FUNCTION_BLOCK PUBLIC ElmoBasicAxis_FB EXTENDS CoE_BasicAxis_FB  
VAR_INPUT		
	pDigIn: 		    POINTER TO DINT;
	
END_VAR
VAR_IN_OUT	
END_VAR
VAR_OUTPUT	
END_VAR

VAR
	
	fbElmoIOsHandle:	FB_ElmoIOsHandle;
END_VAR


AxisCtrlPtr^.Input.Parameter.Drive.eDriveType := enumDriveType.eElmo;	
AxisCtrlPtr^.Input.Parameter.Drive.VendorNameID := eVendorNameID.Elmo;
SUPER^(AxisRef:=AxisRef);


IF pDigIn <> 0 THEN
	fbElmoIOsHandle(DigIn:=	pDigIn^);
	AxisCtrlPtr^.Output.Status.DriveEnable:=	fbElmoIOsHandle.bEnable;
END_IF

METHOD CreateDriveErrMsgDetails : enumMotorEvents
VAR_INPUT
	ErrorId			: UDINT;
END_VAR
CASE ErrorId OF
	16#0:
		CreateDriveErrMsgDetails := enumMotorEvents.NoEvents;
		
	16#2340:
		CreateDriveErrMsgDetails := enumMotorEvents.MotorSupplyError;
		fnLogMsg(ADR(LogMsg_0),LOG_ERROR,'Elmo Drive ErrorId %d  ,Short circuit',UDINT_TO_DINT(ErrorId),0,0);
	16#3120: 
		CreateDriveErrMsgDetails := enumMotorEvents.MotorSupplyError;
		fnLogMsg(ADR(LogMsg_0),LOG_ERROR,'Elmo Drive ErrorId %d Under Voltage',UDINT_TO_DINT(ErrorId),0,0);
	16#3130:
		CreateDriveErrMsgDetails := enumMotorEvents.MotorSupplyError;
		fnLogMsg(ADR(LogMsg_0),LOG_ERROR,'Elmo Drive ErrorId %d Hall  AC fail,loss off phase',UDINT_TO_DINT(ErrorId),0,0);
	16#3310:
		CreateDriveErrMsgDetails := enumMotorEvents.MotorOverCurrent ;
		fnLogMsg(ADR(LogMsg_0),LOG_ERROR,' voltage is too high',UDINT_TO_DINT(ErrorId),0,0);
 
	16#4310:
		CreateDriveErrMsgDetails := enumMotorEvents.MotorOverTemp ;
		fnLogMsg(ADR(LogMsg_0),LOG_ERROR,'Elmo Drive ErrorId %d Temp drive overhating',UDINT_TO_DINT(ErrorId),0,0);
	16#5280:
		CreateDriveErrMsgDetails := enumMotorEvents.MotorPositionError ;	
		fnLogMsg(ADR(LogMsg_0),LOG_ERROR,'Elmo Drive ErrorId %d Gantry position error',UDINT_TO_DINT(ErrorId),0,0);
		
	16#5441:
		CreateDriveErrMsgDetails := enumMotorEvents.DriveNotEnabled;
		fnLogMsg(ADR(LogMsg_0),LOG_ERROR,'Elmo Drive ErrorId %d Motor disables',UDINT_TO_DINT(ErrorId),0,0);
	16#5442:
		CreateDriveErrMsgDetails := enumMotorEvents.DriveNotEnabled;
		fnLogMsg(ADR(LogMsg_0),LOG_ERROR,'Elmo Drive ErrorId %d Motor disables by sw',UDINT_TO_DINT(ErrorId),0,0);
	16#6300:
		CreateDriveErrMsgDetails := enumMotorEvents.PLCIllegalParam;
		fnLogMsg(ADR(LogMsg_0),LOG_ERROR,'Elmo Drive ErrorId %d RPDO failed',UDINT_TO_DINT(ErrorId),0,0);
	16#7121:
		CreateDriveErrMsgDetails := enumMotorEvents.MotorPositionError;
		fnLogMsg(ADR(LogMsg_0),LOG_ERROR,'Elmo Drive ErrorId %d Motor stuck',UDINT_TO_DINT(ErrorId),0,0);
	16#7300:
		CreateDriveErrMsgDetails := enumMotorEvents.MotorFeedBackErr;
		fnLogMsg(ADR(LogMsg_0),LOG_ERROR,'Elmo Drive ErrorId %d Feedback error',UDINT_TO_DINT(ErrorId),0,0);
	16#7381:
 		CreateDriveErrMsgDetails := enumMotorEvents.DriveComError;
		fnLogMsg(ADR(LogMsg_0),LOG_ERROR,'Elmo Drive ErrorId %d 2 Dig halls sens where cng on the same time',UDINT_TO_DINT(ErrorId),0,0);
	16#7382: 
		CreateDriveErrMsgDetails := enumMotorEvents.MotorPositionError;
		fnLogMsg(ADR(LogMsg_0),LOG_ERROR,'Elmo Drive ErrorId %d Commutaition procees failed',UDINT_TO_DINT(ErrorId),0,0);
	16#8110:
		CreateDriveErrMsgDetails := enumMotorEvents.DriveComError;
		fnLogMsg(ADR(LogMsg_0),LOG_ERROR,'Elmo Drive ErrorId %d Cam Msg lost',UDINT_TO_DINT(ErrorId),0,0);
	16#8130:
		CreateDriveErrMsgDetails := enumMotorEvents.DriveComError;
		fnLogMsg(ADR(LogMsg_0),LOG_ERROR,'Elmo Drive ErrorId %d Heartbeat event',UDINT_TO_DINT(ErrorId),0,0);
	16#8140:
		CreateDriveErrMsgDetails := enumMotorEvents.MotorGeneralError;
		fnLogMsg(ADR(LogMsg_0),LOG_ERROR,'Elmo Drive ErrorId %d Recovered from bus off',UDINT_TO_DINT(ErrorId),0,0);
	16#8210:
		CreateDriveErrMsgDetails := enumMotorEvents.MotorGeneralError;
		fnLogMsg(ADR(LogMsg_0),LOG_ERROR,'Elmo Drive ErrorId %d access to non configured PDO',UDINT_TO_DINT(ErrorId),0,0);
	16#8311:
		CreateDriveErrMsgDetails := enumMotorEvents.MotorOverCurrent;
		fnLogMsg(ADR(LogMsg_0),LOG_ERROR,'Elmo Drive ErrorId %d Peak current has been exceeded',UDINT_TO_DINT(ErrorId),0,0);

	16#8480:
		CreateDriveErrMsgDetails := enumMotorEvents.MotorSpeedError;
		fnLogMsg(ADR(LogMsg_0),LOG_ERROR,'Elmo Drive ErrorId %d speed tracking Error',UDINT_TO_DINT(ErrorId),0,0);
	16#8481:
		CreateDriveErrMsgDetails := enumMotorEvents.MotorSpeedError;
		fnLogMsg(ADR(LogMsg_0),LOG_ERROR,'Elmo Drive ErrorId %d Speed limit Exceeded',UDINT_TO_DINT(ErrorId),0,0);
	16#8611:
		CreateDriveErrMsgDetails := enumMotorEvents.MotorPositionError;
		fnLogMsg(ADR(LogMsg_0),LOG_ERROR,'Elmo Drive ErrorId %d Position tracking error',UDINT_TO_DINT(ErrorId),0,0);
	16#8680:
		CreateDriveErrMsgDetails := enumMotorEvents.MotorPositionError;
		fnLogMsg(ADR(LogMsg_0),LOG_ERROR,'Elmo Drive ErrorId %d Position limit Exceeded',UDINT_TO_DINT(ErrorId),0,0);
	16#FF02:
		CreateDriveErrMsgDetails := enumMotorEvents.DriveComError;
		fnLogMsg(ADR(LogMsg_0),LOG_ERROR,'Elmo Drive ErrorId %d Com Error',UDINT_TO_DINT(ErrorId),0,0);
	16#FF10:
		CreateDriveErrMsgDetails := enumMotorEvents.MotorGeneralError ;
		fnLogMsg(ADR(LogMsg_0),LOG_ERROR,'Elmo Drive ErrorId %d Failed to start motor',UDINT_TO_DINT(ErrorId),0,0);
	16#FF20:
		CreateDriveErrMsgDetails := enumMotorEvents.MotorGeneralError;
		fnLogMsg(ADR(LogMsg_0),LOG_ERROR,'Elmo Drive ErrorId %d Saftey torque Off in use',UDINT_TO_DINT(ErrorId),0,0);
	16#FF40:
		CreateDriveErrMsgDetails := enumMotorEvents.MotorGeneralError;
		fnLogMsg(ADR(LogMsg_0),LOG_ERROR,'Elmo Drive ErrorId %d Gantry slave Disabled',UDINT_TO_DINT(ErrorId),0,0);
	ELSE
		fnLogMsg(ADR(LogMsg_0),LOG_ERROR,'unknown Elmo Drive ErrorId %d ',UDINT_TO_DINT(ErrorId),0,0);
		CreateDriveErrMsgDetails := enumMotorEvents.MotorGeneralError;
		 
END_CASE
END_METHOD

METHOD DriveUnitsTorqueToRealValue : LREAL
VAR_INPUT
	
	Torque: LREAL;	

END_VAR
DriveUnitsTorqueToRealValue := (Torque*AxisCtrlPtr^.Input.Parameter.RatedCurrent)/1000;
END_METHOD

METHOD GetCanOpenAdr : BOOL
VAR_INPUT
END_VAR


VAR
	
	SpeedSwSubIndex: INT;
END_VAR
    SUPER^.GetCanOpenAdr();	

	
	CoEDrive_Ctrl_Adr.KpSpeed.Index	   := 16#3113;	
	CoEDrive_Ctrl_Adr.KpSpeed.SunIndex  := 2;
	CoEDrive_Ctrl_Adr.KpSpeed.Size      := 4;
	CoEDrive_Ctrl_Adr.KpSpeed.IsReal    := TRUE;
	
	
	CoEDrive_Ctrl_Adr.KiSpeed.Index	    := 16#310C;	
	CoEDrive_Ctrl_Adr.KiSpeed.SunIndex  := 2;
   	CoEDrive_Ctrl_Adr.KiSpeed.Size      := 4;
	CoEDrive_Ctrl_Adr.KiSpeed.IsReal    := TRUE;
	
	CoEDrive_Ctrl_Adr.GainScheduler.Index	    := 16#30AE;	
	CoEDrive_Ctrl_Adr.GainScheduler.SunIndex    := 2;
   	CoEDrive_Ctrl_Adr.GainScheduler.Size        := 8;
	
	
	CoEDrive_Ctrl_Adr.AccClosePosErr.Index	    := 16#30AE;	
	CoEDrive_Ctrl_Adr.AccClosePosErr.SunIndex    := 9;
   	CoEDrive_Ctrl_Adr.AccClosePosErr.Size        := 8;
END_METHOD

METHOD GetErrCanAdr : BOOL
VAR_INPUT
END_VAR


VAR
	
END_VAR

	
	CoeErrIdIndex	 := 16#603F;
	CoeErrIdSubIndex := 0;
END_METHOD

METHOD  INIT_Specific : BOOL 
VAR_INPUT
	bStart: 					BOOL;
END_VAR
VAR_INST	
	ComDelay:	TON;
	Elmo_Init_State : INT ;
	ExecuteTrig: 	Trigger;
END_VAR
IF ExecuteTrig.EDGEPOS(bStart) THEN
	INIT_Specific := FALSE ;
	IF AxisCtrlPtr^.Input.Parameter.Drive.bDisableFoE_Transfer THEN 
		Elmo_Init_State:= 3;
	ELSE
		CoEDrive_Ctrl_Adr.ParamsVersionObj.Index    := 16#2F00;
		CoEDrive_Ctrl_Adr.ParamsVersionObj.SunIndex := 1; 		
		Elmo_Init_State:= 1;
	END_IF
END_IF


IF ExecuteTrig.EDGENEG(bStart) THEN
	Elmo_Init_State := 0;
END_IF	

	
CASE Elmo_Init_State OF							
	1:
		Meth_UpdateDriveParams(FALSE);
		Elmo_Init_State:=	2;
	2:	
		IF Meth_UpdateDriveParams(TRUE) THEN
			Elmo_Init_State:=	3;
		ELSIF AxisCtrlPtr^.Output.Status.Drive.eUpdate_Staus = enum_DriveUpdateStatus.Error THEN
			//
		END_IF

	3:
		ReadInitDriveParID(FALSE);
		Elmo_Init_State:=	4;
		
	4:
		IF ReadInitDriveParID(TRUE) THEN
			Elmo_Init_State:=	10;
		END_IF			

	10:
		
		Elmo_Init_State := 0 ;
		INIT_Specific := TRUE ;
		AxisCtrlPtr^.Output.Status.AxisInitDone := TRUE ;
		AxisCtrlPtr^.Output.Status.ReadyForCmd := TRUE ;
END_CASE
END_METHOD

METHOD Meth_ChangingOperationMode : BOOL
VAR_INPUT
	Execute   : BOOL;
	OperMode : eDriveModeOfOperation; 
	
END_VAR
VAR_INST
	
	ElmoCngOperState : INT;	
END_VAR

VAR
	
	ChangeDone : BOOL;
END_VAR
IF ChangeModeOperTrig.EDGEPOS(Execute) THEN

	Meth_ChangingOperationMode := FALSE;					
	ChangeDone := FALSE;
	ElmoCngOperState := 1;

	
END_IF


IF ChangeModeOperTrig.EDGENEG(Execute) THEN
	
	ElmoCngOperState := 0;
END_IF



CASE ElmoCngOperState OF
	0:
		Meth_CoEChangOperationMode(FALSE,eCaOpDriveModeOfOperation.ProfilePositionMode);
		
	1: 
		//Meth_CoEChangOperationMode
		CASE OperMode OF
			eDriveModeOfOperation.ProfilePositionMode				:
				IF Meth_CoEChangOperationMode(TRUE,eCaOpDriveModeOfOperation.ProfilePositionMode) THEN
					ChangeDone := TRUE;
				END_IF
				
		    eDriveModeOfOperation.VelocityCtrMode    				:
				IF Meth_CoEChangOperationMode(TRUE,eCaOpDriveModeOfOperation.ProfileVelocityMode)THEN
					ChangeDone := TRUE;
				END_IF
		    eDriveModeOfOperation.ProfileVelocityMode 	   	    :
				IF Meth_CoEChangOperationMode(TRUE,eCaOpDriveModeOfOperation.ProfileVelocityMode) THEN
					ChangeDone := TRUE;
				END_IF
				
		    eDriveModeOfOperation.TorqueVelocityMode 				:
				IF Meth_CoEChangOperationMode(TRUE,eCaOpDriveModeOfOperation.TorqueVelocityMode) THEN
					ChangeDone := TRUE;
				END_IF
				
		    eDriveModeOfOperation.HomingMode				    	:
				IF Meth_CoEChangOperationMode(TRUE,eCaOpDriveModeOfOperation.HomingMode)THEN
					ChangeDone := TRUE;
				END_IF
				
		    eDriveModeOfOperation.InterpolationPosMode			:
				IF Meth_CoEChangOperationMode(TRUE,eCaOpDriveModeOfOperation.InterpolationPosMode) THEN
					ChangeDone := TRUE;
				END_IF
		    eDriveModeOfOperation.CyclicSyncMode					:
				Meth_CoEChangOperationMode(TRUE,eCaOpDriveModeOfOperation.CyclicSyncMode);
		END_CASE
		ElmoCngOperState := 2;

	2:
 		Meth_ChangingOperationMode := TRUE;
		
		
END_CASE
END_METHOD

METHOD Meth_TorqueInDriveUnits : LREAL
VAR_INPUT
	
	Torque: LREAL;	

END_VAR
IF AxisCtrlPtr^.Input.Parameter.RatedCurrent <> 0 THEN
	Meth_TorqueInDriveUnits := (Torque*1000)/AxisCtrlPtr^.Input.Parameter.RatedCurrent;
END_IF
END_METHOD

METHOD ReadActualCurrent : LREAL
VAR_INPUT
END_VAR
VAR_INST
		
END_VAR


// Units [rms]

AxisCtrlPtr^.Output.monitor.ActualCurrent	:=  ( (THIS^.io_ActualCurrent) / 1000.0) * AxisCtrlPtr^.Input.Parameter.RatedCurrent / SQRT(2.0);
END_METHOD

METHOD ReadActualTorque : LREAL
VAR_INPUT
END_VAR
VAR_INST
		
END_VAR

// Units [rms]
//AxisCtrlPtr^.Output.monitor.ActualCurrent Get from ReadActualCurrent method
// on Elmo it is needed to link only IO  io_ActualCurrent
AxisCtrlPtr^.Output.monitor.ActualTorque	:=  AxisCtrlPtr^.Output.monitor.ActualCurrent * AxisCtrlPtr^.Input.Parameter.Drive.Kt;
END_METHOD

METHOD ReadInitDriveParID : BOOL
VAR_INPUT
	bStart : BOOL;
END_VAR

VAR_INST
	ExecuteTrig_1: 		Trigger;
	State_InitSpecific_1: INT;
END_VAR

IF ExecuteTrig_1.EDGEPOS(bStart) THEN
	ReadInitDriveParID		:= FALSE;
	State_InitSpecific_1	:= 1;		
END_IF

IF ExecuteTrig_1.EDGENEG(bStart) THEN
	State_InitSpecific_1	:= 0;	
	ReadInitDriveParID		:= FALSE;
END_IF

CASE State_InitSpecific_1 OF

	 
	
	1:
		SUPER^.EcCoeSdoRead(FALSE);
		CoeSdoRW.Input.Read.nIndex		:= DINT_TO_WORD(eElmoDriveParID.RatedCurrent);
		CoeSdoRW.Input.Read.nSubIndex	:= 0;
		CoeSdoRW.Input.Read.pDstBuf		:= ADR(CoeRead_RatedCurrent);
		CoeSdoRW.Input.Read.cbBufLen	:= SIZEOF(CoeRead_RatedCurrent);
		State_InitSpecific_1	:= 2;
		
	2:
		IF SUPER^.EcCoeSdoRead(TRUE) THEN	
			State_InitSpecific_1	:= 3;
		END_IF
		
	3:
		SUPER^.EcCoeSdoRead(FALSE);
		CoeSdoRW.Input.Read.nIndex		:= DINT_TO_WORD(eElmoDriveParID.RatedTorque);
		CoeSdoRW.Input.Read.nSubIndex	:= 0;
		CoeSdoRW.Input.Read.pDstBuf		:= ADR(CoeRead_RatedTorque);
		CoeSdoRW.Input.Read.cbBufLen	:= SIZEOF(CoeRead_RatedTorque);
		State_InitSpecific_1	:= 4;
		
	4:
		IF SUPER^.EcCoeSdoRead(TRUE) THEN
			AxisCtrlPtr^.Input.Parameter.RatedCurrent	:= UDINT_TO_LREAL(CoeRead_RatedCurrent) / 1000.0;
			AxisCtrlPtr^.Input.Parameter.Ratedtorque	:= UDINT_TO_LREAL(CoeRead_RatedTorque) / 1000.0;
			ReadInitDriveParID		:= TRUE;	
			State_InitSpecific_1	:= 0;
		END_IF
		
END_CASE
END_METHOD

END_FUNCTION_BLOCK

(* stored: Version 1.1.0.1, ProductVersion 3.1.4024.3
   POU ElmoBasicAxis_FB: Id {2e0e12a1-cbda-0a39-099b-5ee932b872e2}, SpecialFunc None
   Method CreateDriveErrMsgDetails: Id {9cc976e0-d151-0c3a-0286-72b050a07b1d}
   Method DriveUnitsTorqueToRealValue: Id {655fd303-8479-4aac-a951-a73c4774eb58}
   Method GetCanOpenAdr: Id {5459baee-fb42-4764-b410-c7c8356edfd8}
   Method GetErrCanAdr: Id {87d06868-b33e-0803-257c-791b5bbbc79f}
   Method INIT_Specific: Id {ff4c39ef-11b0-019e-39fa-a81d964c7711}
   Method Meth_ChangingOperationMode: Id {335ef2a7-70a9-4328-9a4c-78491bccc262}
   Method Meth_TorqueInDriveUnits: Id {0b404ad3-f140-4a59-b6f1-dbfb474491a6}
   Method ReadActualCurrent: Id {e92bc553-4eb8-43f0-9e6c-04388d0f3070}
   Method ReadActualTorque: Id {703882d2-916f-4ffe-8cd7-2ccba07b8635}
   Method ReadInitDriveParID: Id {cfd5b54e-9c59-48c8-9b20-0b19b3d9d026} *)
